GLOBALCONSTANTS START (* START States *)
  (* Standard: 61499-1; Description: Copyright (c) 2025 HR Agrartechnik GmbH This program and the accompanying materials are made available under the terms of the Eclipse Public License 2.0 which is available at https://www.eclipse.org/legal/epl-2.0/ SPDX-License-Identifier: EPL-2.0 *)
  (* Version 1.0, 2025-05-23, Franz Höpfinger, HR Agrartechnik GmbH *)
  PACKAGE logiBUS::utils::sequence::schieber::const;
  IMPORT eclipse4diac::core::TypeHash;
  VAR_GLOBAL CONSTANT
    STARTClosed : UINT := UINT#5;
    STARTOpened : UINT := UINT#6;
    STARTUnknown : UINT := UINT#7;
  END_VAR
END_GLOBALCONSTANTS
